INTERFACE I_RequestHeader

METHOD PUBLIC TryGetField : BOOL;
VAR_INPUT
	Key : STRING;
	Destination : ANY;
END_VAR
END_METHOD

METHOD PUBLIC TryWriteField : BOOL;
VAR_INPUT
	Key : STRING;
	Source : ANY;
END_VAR
END_METHOD

END_INTERFACE

(* stored: Version 1.1.0.1, ProductVersion 3.1.4024.12
   Itf I_RequestHeader: Id {4cde2aee-558d-4169-b9eb-87b201e0fad0}
   Method TryGetField: Id {a07cba59-e882-4def-8d2a-5f95e635fa70}
   Method TryWriteField: Id {6b520cc5-e54a-49f3-9de4-53d1fb1e95ea} *)
